PROGRAM MAIN
VAR
	counter_x : INT;
	
	vgc_reader : FB_TVGC_ADS;
	gcc_reader : FB_TGCC_ADS;
	
END_VAR

// A counter to confirm that the program is running
counter_x := counter_x + 1;

END_PROGRAM

(* stored: Version 1.1.0.1, ProductVersion 3.1.4024.2
   POU MAIN: Id {445c6c3e-5f54-4453-b203-c04c9319e6f6}, SpecialFunc None *)
